(* IEC 61131-3 sources: PLC-PDAM-Samarinda/Object, 6 files *)

(* ---- tank1.st ---- *)
FUNCTION_BLOCK tank1
VAR_INPUT

END_VAR
VAR_OUTPUT

END_VAR
VAR
	inletValve : switchON;
    outletValve : switchON;

END_VAR

//logic
inletValve(power:= );
inletValve.status;

outletValve(power:= );
inlet

END_FUNCTION_BLOCK

(* ---- tank2.st ---- *)
FUNCTION_BLOCK tankank2
VAR_INPUT

END_VAR
VAR_OUTPUT

END_VAR
VAR

END_VAR

//logic

END_FUNCTION_BLOCK

(* ---- tank3.st ---- *)
FUNCTION_BLOCK tank3
VAR_INPUT

END_VAR
VAR_OUTPUT

END_VAR
VAR

END_VAR

//logic

END_FUNCTION_BLOCK

(* ---- tank4.st ---- *)
FUNCTION_BLOCK tank4
VAR_INPUT

END_VAR
VAR_OUTPUT

END_VAR
VAR

END_VAR

//logic

END_FUNCTION_BLOCK

(* ---- tank5.st ---- *)
FUNCTION_BLOCK tank5
VAR_INPUT

END_VAR
VAR_OUTPUT

END_VAR
VAR

END_VAR

//logic

END_FUNCTION_BLOCK

(* ---- tank6.st ---- *)
FUNCTION_BLOCK tank6
VAR_INPUT

END_VAR
VAR_OUTPUT

END_VAR
VAR

END_VAR

//logic

END_FUNCTION_BLOCK
